FUNCTION_BLOCK FB_Component_TE2 EXTENDS FB_BaseComponent IMPLEMENTS ITF_Component_TE2, ITF_Component_TE2_HMI_Init
VAR
END_VAR

METHOD testMethod : BOOL
VAR_INPUT
END_VAR
END_METHOD

END_FUNCTION_BLOCK

(* stored: Version 1.1.0.1, ProductVersion 3.1.4024.15
   POU FB_Component_TE2: Id {b20d8b47-3886-4b8b-b836-316be1a8d7b8}, SpecialFunc None
   Method testMethod: Id {4b9e12f3-f334-4ea3-9195-5df56108187b} *)
